Staubli VAL3: ImpedCtrlTest.dtx

mdesc mNomSpeed
public bool bOverRun = true
public num nMass[6 6]
  [0,0] = 1
  [1,1] = 1
  [2,2] = 1
  [3,3] = 1
  [4,4] = 1
  [5,5] = 1
public num nStiffness[6 6]
  [0,0] = 25
  [1,1] = 25
  [2,2] = 25
  [3,3] = 25
  [4,4] = 25
  [5,5] = 25
public num nDamp[6 6]
  [0,0] = 10
  [1,1] = 10
  [2,2] = 10
  [3,3] = 10
  [4,4] = 10
  [5,5] = 10
public num ndForce[6]
public num ndAccel[6]
public num ndVelocity[6]
public num nForce[6]
public num ndPosition[6]
public mdesc mImpedSpeed = {blend=off}
public pointRx pNowPosition = {fatherId=world[0]}
public num nNowVelocity[6]
public num nNowAccel[6]
public num nLastVelocity[6]
public num nNowClock
public num nTime
public sio sClient = {link=Socket\FTSensor}
public num nForceTorque[6]
  [0] = -0.458435
  [1] = -0.0611247
  [2] = -0.0305157
  [3] = 0.00182448
  [4] = 0.00243784
public num nPort = 5001
public num nSensitivity[6]
  [0] = 32.72
  [1] = 32.72
  [2] = 32.77
  [3] = 1644.3
  [4] = 1640.8
  [5] = 1635
public num nSioTimeOut = 5
public num nZeroPoint[6]
  [0] = 8211
  [1] = 8189
  [2] = 8176
  [3] = 8194
  [4] = 8176
  [5] = 8189
public pointRx pCommand = {fatherId=world[0]}
